// Deallocates memory associated with a generic value and resets it to a default state.
FUNCTION F_DeallocateGeneric
VAR_IN_OUT
	Value : FsCommon.T_Generic; // The generic value whose memory will be deallocated.
END_VAR

FsCommon.F_DeallocateMemory(Value.pValue);
Value.diSize := 0;
Value.TypeClass := __SYSTEM.TYPE_CLASS.TYPE_NONE;

END_FUNCTION

(* stored: Version 1.1.0.1
   POU F_DeallocateGeneric: Id {4b979afb-b3a9-0286-064d-8d769ea4ee90}, SpecialFunc None *)
